FUNCTION Convert_TIME_TO_TOD : Hresult
VAR_INPUT
	in : TIME;
	out : REFERENCE TO TOD;
END_VAR
VAR
	converted : TOD;
END_VAR

converted := TIME_TO_TOD(in);

IF (TOD_TO_TIME(converted) <> in) THEN
	Convert_TIME_TO_TOD := INCOMPATIBLE;
	RETURN;
END_IF

out := converted;

END_FUNCTION

(* stored: Version 1.1.0.1, ProductVersion 3.1.4024.12
   POU Convert_TIME_TO_TOD: Id {f223a114-03a3-47bb-893c-82dae2a96b94}, SpecialFunc None *)
